FUNCTION SelectMovement : BYTE
VAR_INPUT
	ManualMode: BOOL;
END_VAR
VAR
	MovementSelection: CTUD;
	SelectionCounter: CTUD := (LOAD := TRUE, PV := 3);
	ReachedMaxSelection: BOOL;
	ReachedMinSelection: BOOL;
END_VAR
VAR_OUTPUT
	CurrentSelection: INT;
END_VAR

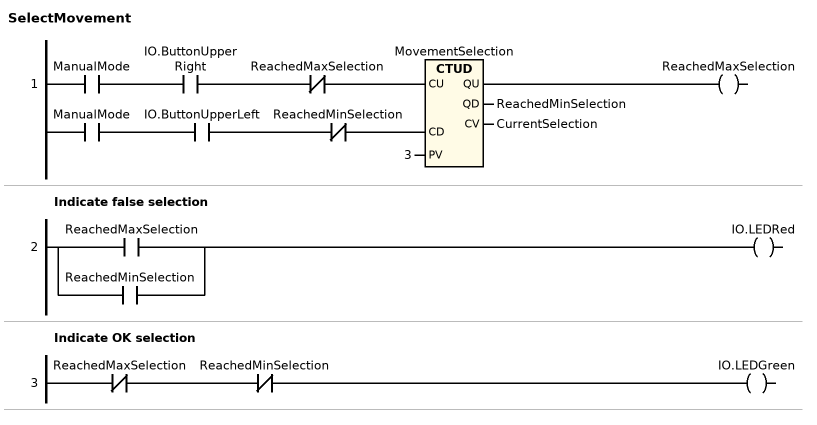
// NETWORK 1
MovementSelection(
    CU := ManualMode AND IO.ButtonUpperRight AND NOT ReachedMaxSelection,
    CD := ManualMode AND IO.ButtonUpperLeft AND NOT ReachedMinSelection,
    PV := 3,
    QD => ReachedMinSelection,
    CV => CurrentSelection); // CTUD
ReachedMaxSelection := MovementSelection.QU;

// NETWORK 2: Indicate false selection
IO.LEDRed := ReachedMaxSelection OR ReachedMinSelection;

// NETWORK 3: Indicate OK selection
IO.LEDGreen := NOT ReachedMaxSelection AND NOT ReachedMinSelection;

END_FUNCTION

(* stored: Version 1.1.0.1, ProductVersion 3.1.4024.13
   POU SelectMovement: Id {b5b93571-81d8-404e-937f-9acd97ccf1e3}, SpecialFunc None *)
